// TIA Portal V19 export
DATA_BLOCK "DB_BE_Stand"   // DB4
{ S7_Optimized_Access := 'FALSE' }
// stored: AutoNumber false
   VAR RETAIN
      Anzahl : Int := 6;   // * Anzahl der BE-/Entladestände
      leng : Int := 12;   // * Länge einer Struktur
      Offset : Int := 10;   // * Beginn des Datenfeldes
      Next : Byte := 16#00;   // nächster Wt für die Anlage
      Entm : Byte := 16#00;   // nächster Wt für die Entmetallisierung
      AnfQ : Byte := 16#00;   // Anforderung Quelle
      AnfZ : Byte := 16#00;   // Anforderung Ziel
      Stand : Array[1..6] of Struct   // * Feldlänge anpassen
         Pos_Nr : USInt;
         Aufgabe_erlaubt : Bool;   // Aufgabe ist möglich
         kein_WT : Bool;   // Stand ist leer (WT ist weder physikalisch noch logisch vorhanden)
         WT_aufgegeben : Bool;   // Warenträger ist aufgegeben
         verriegelt : Bool;   // Bedienung durch FW möglich
         gelb : Bool;
         rot : Bool;
         Charge_ok : Bool;   // Behandlung war fehlerfrei
         Charge_nok : Bool;   // Behandlung war gestört
         IN_innen : Bool;   // Wagen angedockt
         IN_aussen : Bool;   // Wagen im Beladebereich
         IN_Belegt : Bool;   // WT auf Wagen
         IN_Freigabe : Bool;   // Freigabetaste (wennvorhanden über Flankenmerker Bit4.0)
         OUT_Sperre_in : Bool;   // Einfahrsperre
         OUT_Sperre_FW : Bool;   // Überfahrsperre
         OUT_Sperre_out : Bool;   // Ausfahrsperre
         OUT_FW_kommt : Bool;   // Meldung FW kommt
         Del_Count : Byte;   // Sekundenzähler zum löschen der WT-Info
         AM_Freigabe : Bool;   // Altmerker Freigabetaste
         AM_Wagen : Bool;   // Altmerker Wagen vorhanden
         res3 : Bool;
         Trommel_BE : Bool;   // Trommelstand
         Gestell_BE : Bool;   // Gestellstand
         Ausf_Ware : Bool;   // Ausfahrt Ware erlaubt
         Ausf_Entm : Bool;   // Ausfahrt entmetallisierte Gestelle
         last_WT_Trommel : Bool;   // letzter WT war / ist Trommel
         Anf_Pos : Byte;   // Position die BE-Anfordert
         last_WT : DInt;   // letzte WT-Nr-lang
         Del_All : Bool;   // 0=Programm löschen 1=gesamten WT löschen
         Auto_Delete : Bool;   // automatisches löschen fertiger WT
         Afg_WT_Nr : Bool;   // Aufgabe auch bei WT_Nr_lang<>0 erlaubt
         res1 : Bool;
         res2 : Bool;
         res4 : Bool;
         res5 : Bool;
         schnell : Bool;
         resB : Byte;
      END_STRUCT;
      Langware_vorn : Bool;
      Langware_hinten : Bool;
   END_VAR
BEGIN
   Stand[1].Pos_Nr := 25;
   Stand[2].Pos_Nr := 26;
   Stand[3].Pos_Nr := 27;
   Stand[4].Pos_Nr := 28;
   Stand[5].Pos_Nr := 29;
   Stand[6].Pos_Nr := 30;
   Stand[1..5].Aufgabe_erlaubt := FALSE;
   Stand[1..3].kein_WT := TRUE;
   Stand[4..5].kein_WT := FALSE;
   Stand[1..5].WT_aufgegeben := FALSE;
   Stand[1].verriegelt := FALSE;
   Stand[2].verriegelt := TRUE;
   Stand[3..5].verriegelt := FALSE;
   Stand[1..5].gelb := FALSE;
   Stand[1..5].rot := FALSE;
   Stand[1..5].Charge_ok := FALSE;
   Stand[1..5].Charge_nok := FALSE;
   Stand[1].IN_innen := FALSE;
   Stand[2].IN_innen := TRUE;
   Stand[3..5].IN_innen := FALSE;
   Stand[1].IN_aussen := FALSE;
   Stand[2].IN_aussen := TRUE;
   Stand[3..5].IN_aussen := FALSE;
   Stand[1..5].IN_Belegt := FALSE;
   Stand[1].IN_Freigabe := FALSE;
   Stand[2].IN_Freigabe := TRUE;
   Stand[3..5].IN_Freigabe := FALSE;
   Stand[1].OUT_Sperre_in := TRUE;
   Stand[2..5].OUT_Sperre_in := FALSE;
   Stand[1..5].OUT_Sperre_FW := FALSE;
   Stand[1..2].OUT_Sperre_out := TRUE;
   Stand[3..5].OUT_Sperre_out := FALSE;
   Stand[1..5].OUT_FW_kommt := FALSE;
   Stand[1].Del_Count := 16#05;
   Stand[2].Del_Count := 16#1E;
   Stand[3..5].Del_Count := 16#00;
   Stand[1..5].AM_Freigabe := FALSE;
   Stand[1..2].AM_Wagen := TRUE;
   Stand[3..5].AM_Wagen := FALSE;
   Stand[1..5].res3 := FALSE;
   Stand[1..5].Trommel_BE := FALSE;
   Stand[1..5].Gestell_BE := FALSE;
   Stand[1..5].Ausf_Ware := FALSE;
   Stand[1..5].Ausf_Entm := FALSE;
   Stand[1..5].last_WT_Trommel := FALSE;
   Stand[1..5].Anf_Pos := 16#00;
   Stand[1..5].last_WT := 0;
   Stand[1..2].Del_All := TRUE;
   Stand[3..5].Del_All := FALSE;
   Stand[1].Auto_Delete := FALSE;
   Stand[2].Auto_Delete := TRUE;
   Stand[3..5].Auto_Delete := FALSE;
   Stand[1..5].Afg_WT_Nr := FALSE;
   Stand[1..5].res1 := FALSE;
   Stand[1..5].res2 := FALSE;
   Stand[1..5].res4 := FALSE;
   Stand[1..5].res5 := FALSE;
   Stand[1..5].schnell := FALSE;
   Stand[1..5].resB := 16#00;
END_DATA_BLOCK
